// TIA Portal project "SemaforV1" (V15.1)

(* hardware
DEVICE "S71500/ET200MP station_1"  S7-1500 station
   slot 0: "Rail_0"  Rack  6ES7 590-1***0-0AA0
   slot 1: "PLC_1"  CPU 1513-1 PN  6ES7 513-1AL02-0AB0  V2.6
      slot 3: "CPU display_1"  6ES7591-1AA00-0AA0
DEVICE "HMI_1"  KTP900 Basic PN
   slot 0: "HMI_1"  KTP900 Basic PN  6AV2 123-2JB03-0AX0  15.1.0.0
   slot 1: "HMI_RT_1"  KTP900 Basic PN  6AV2 123-2JB03-0AX0  15.1.0.0
   slot 5: "HMI_1.IE_CP_1"  PROFINET Interface  15.0.1.0
      slot 1: "PROFINET Interface_1"  PROFINET Interface
         slot 1: "Port_1"  Port
*)

// ===== PLC "PLC_1"  CPU 1513-1 PN =====

VAR_GLOBAL   // PLC tag table "Default tag table"
   "Clock_Byte" AT %MB0 : Byte;
   "Clock_10Hz" AT %M0.0 : Bool;
   "Clock_5Hz" AT %M0.1 : Bool;
   "Clock_2.5Hz" AT %M0.2 : Bool;
   "Clock_2Hz" AT %M0.3 : Bool;
   "Clock_1.25Hz" AT %M0.4 : Bool;
   "Clock_1Hz" AT %M0.5 : Bool;
   "Clock_0.625Hz" AT %M0.6 : Bool;
   "Clock_0.5Hz" AT %M0.7 : Bool;
END_VAR

DATA_BLOCK "Semafor_Lumini"   // DB1
{ S7_Optimized_Access := 'TRUE' }
VERSION : 0.1
   VAR
      rosu_on : Bool;
      galben_on : Bool;
      verde_on : Bool;
      culoare_semafor : UInt;
      galben_intermitent_on : Bool;
   END_VAR
BEGIN
END_DATA_BLOCK

DATA_BLOCK "Semafor_Moduri"   // DB2
{ S7_Optimized_Access := 'TRUE' }
VERSION : 0.1
   VAR
      "mod_de functionare" : UInt;
      pornire_mod_normal : Bool;
      reseteaza_bucla : Bool;
      porneste_verde : Bool;
      porneste_galben : Bool;
      porneste_rosu : Bool;
      buton_pieton : Bool;
      timp_rosu : Time;
      Timp_galben : Time;
      timp_verde : Time;
      et_rosu : Time;
      et_galben : Time;
      et_verde : Time;
      timer_galben_hmi : Bool;
   END_VAR
BEGIN
END_DATA_BLOCK

DATA_BLOCK "Rising Edges"   // DB3
{ S7_Optimized_Access := 'TRUE' }
VERSION : 0.1
   VAR
      re1 : Bool;
      testing : Bool;
      "test count" : UInt;
   END_VAR
BEGIN
END_DATA_BLOCK

// folder: System blocks/Program resources

DATA_BLOCK "timer_verde"   // DB4
{ S7_Optimized_Access := 'TRUE' }
AUTHOR : Simatic
FAMILY : IEC
NAME : IEC_TMR
VERSION : 1.0
// stored: InstanceOfName IEC_TIMER
"IEC_TIMER"
BEGIN
END_DATA_BLOCK

DATA_BLOCK "timergalben"   // DB5
{ S7_Optimized_Access := 'TRUE' }
AUTHOR : Simatic
FAMILY : IEC
NAME : IEC_TMR
VERSION : 1.0
// stored: InstanceOfName IEC_TIMER
"IEC_TIMER"
BEGIN
END_DATA_BLOCK

DATA_BLOCK "timer rosu"   // DB6
{ S7_Optimized_Access := 'TRUE' }
AUTHOR : Simatic
FAMILY : IEC
NAME : IEC_TMR
VERSION : 1.0
// stored: InstanceOfName IEC_TIMER
"IEC_TIMER"
BEGIN
END_DATA_BLOCK

// folder: (top level)

ORGANIZATION_BLOCK "Main"   // OB1, LAD, ProgramCycle
TITLE = "Main Program Sweep (Cycle)"
{ S7_Optimized_Access := 'TRUE' }
VERSION : 0.1
   VAR_INPUT
      Initial_Call : Bool;   // Initial call of this OB
      Remanence : Bool;   // =True, if remanent data are available
   END_VAR
   VAR_TEMP   // added for the SCL form of the ladder/FBD networks
      _w1 : Bool;
   END_VAR
BEGIN

REGION Network 1: semafor modul normal
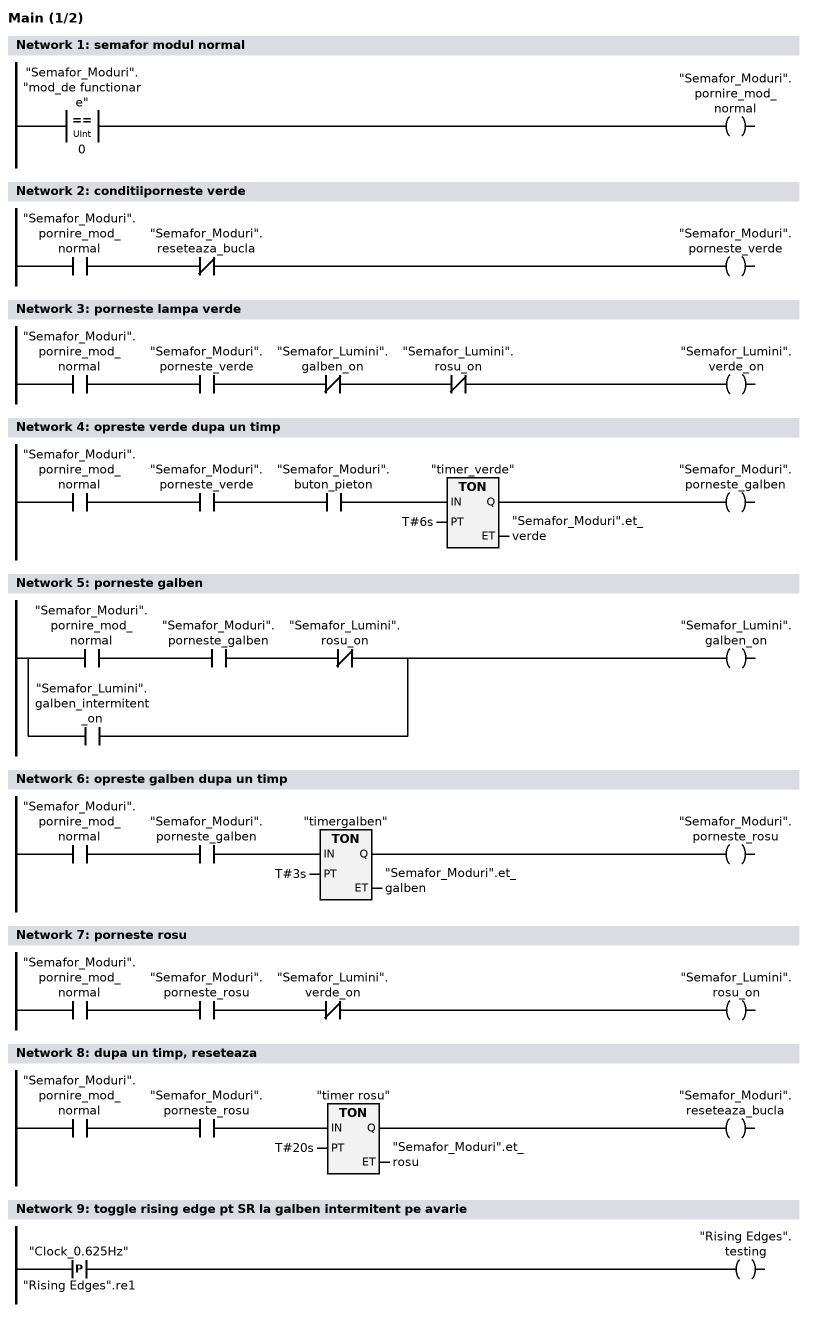
   RUNG wire#powerrail
      { S7_Templates := "SrcType := UInt" } EQ_Contact(in1 := "Semafor_Moduri"."mod_de functionare", in2 := 0)
      Coil( "Semafor_Moduri".pornire_mod_normal )
   END_RUNG
   // the same network as SCL:
   "Semafor_Moduri".pornire_mod_normal := "Semafor_Moduri"."mod_de functionare" = 0;
END_REGION

REGION Network 2: conditiiporneste verde
   RUNG wire#powerrail
      Contact( "Semafor_Moduri".pornire_mod_normal )
      I_Contact( "Semafor_Moduri".reseteaza_bucla )
      Coil( "Semafor_Moduri".porneste_verde )
   END_RUNG
   // the same network as SCL:
   "Semafor_Moduri".porneste_verde := "Semafor_Moduri".pornire_mod_normal AND NOT "Semafor_Moduri".reseteaza_bucla;
END_REGION

REGION Network 3: porneste lampa verde
   RUNG wire#powerrail
      Contact( "Semafor_Moduri".pornire_mod_normal )
      Contact( "Semafor_Moduri".porneste_verde )
      I_Contact( "Semafor_Lumini".galben_on )
      I_Contact( "Semafor_Lumini".rosu_on )
      Coil( "Semafor_Lumini".verde_on )
   END_RUNG
   // the same network as SCL:
   "Semafor_Lumini".verde_on := "Semafor_Moduri".pornire_mod_normal AND "Semafor_Moduri".porneste_verde AND NOT "Semafor_Lumini".galben_on AND NOT "Semafor_Lumini".rosu_on;
END_REGION

REGION Network 4: opreste verde dupa un timp
   "timer_verde".TON(IN := "Semafor_Moduri".pornire_mod_normal AND "Semafor_Moduri".porneste_verde AND "Semafor_Moduri".buton_pieton,
                     PT := T#6s,
                     ET => "Semafor_Moduri".et_verde);
   "Semafor_Moduri".porneste_galben := "timer_verde".Q;
END_REGION

REGION Network 5: porneste galben
   RUNG wire#powerrail
      Contact( "Semafor_Moduri".pornire_mod_normal )
      Contact( "Semafor_Moduri".porneste_galben )
      I_Contact( "Semafor_Lumini".rosu_on )
      wire#w1
      Coil( "Semafor_Lumini".galben_on )
   END_RUNG
   RUNG wire#powerrail
      Contact( "Semafor_Lumini".galben_intermitent_on )
   END_RUNG wire#w1
   // the same network as SCL:
   "Semafor_Lumini".galben_on := ("Semafor_Moduri".pornire_mod_normal AND "Semafor_Moduri".porneste_galben AND NOT "Semafor_Lumini".rosu_on) OR "Semafor_Lumini".galben_intermitent_on;
END_REGION

REGION Network 6: opreste galben dupa un timp
   "timergalben".TON(IN := "Semafor_Moduri".pornire_mod_normal AND "Semafor_Moduri".porneste_galben,
                     PT := T#3s,
                     ET => "Semafor_Moduri".et_galben);
   "Semafor_Moduri".porneste_rosu := "timergalben".Q;
END_REGION

REGION Network 7: porneste rosu
   RUNG wire#powerrail
      Contact( "Semafor_Moduri".pornire_mod_normal )
      Contact( "Semafor_Moduri".porneste_rosu )
      I_Contact( "Semafor_Lumini".verde_on )
      Coil( "Semafor_Lumini".rosu_on )
   END_RUNG
   // the same network as SCL:
   "Semafor_Lumini".rosu_on := "Semafor_Moduri".pornire_mod_normal AND "Semafor_Moduri".porneste_rosu AND NOT "Semafor_Lumini".verde_on;
END_REGION

REGION Network 8: dupa un timp, reseteaza
   "timer rosu".TON(IN := "Semafor_Moduri".pornire_mod_normal AND "Semafor_Moduri".porneste_rosu,
                    PT := T#20s,
                    ET => "Semafor_Moduri".et_rosu);
   "Semafor_Moduri".reseteaza_bucla := "timer rosu".Q;
END_REGION

REGION Network 9: toggle rising edge pt SR la galben intermitent pe avarie
   RUNG wire#powerrail
      P_Contact(operand := "Clock_0.625Hz", bit := "Rising Edges".re1)
      Coil( "Rising Edges".testing )
   END_RUNG
   // the same network as SCL:
   #_w1 := "Clock_0.625Hz" AND NOT "Rising Edges".re1;   // rising edge of "Clock_0.625Hz"
   "Rising Edges".re1 := "Clock_0.625Hz";
   "Rising Edges".testing := #_w1;
END_REGION

REGION Network 10: toggle test 2
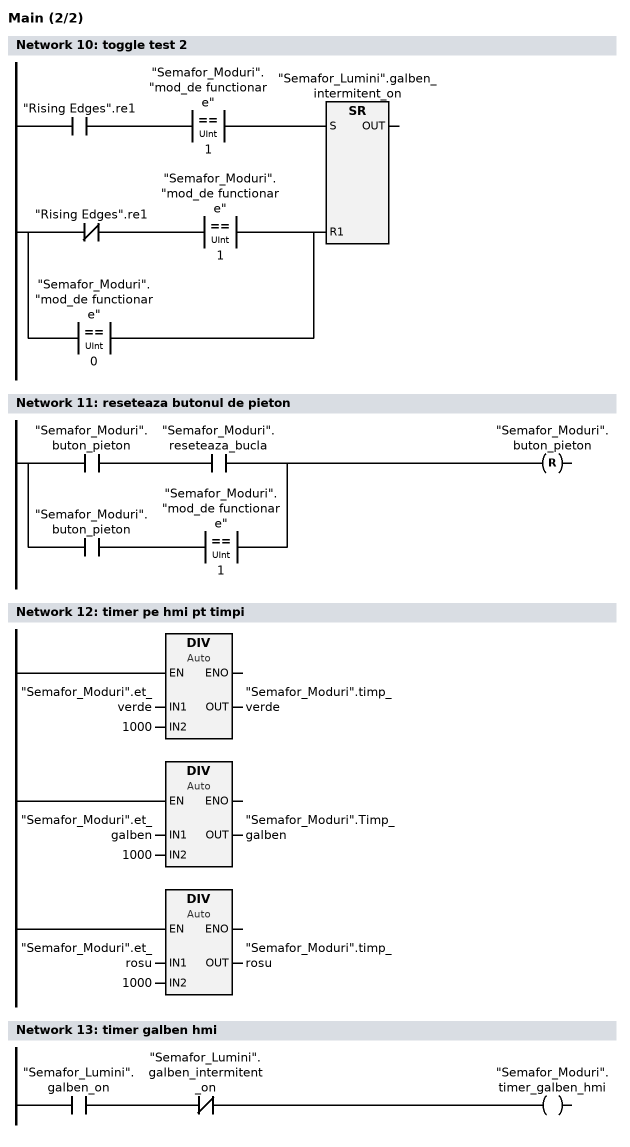
   RUNG wire#powerrail
      Contact( "Rising Edges".re1 )
      { S7_Templates := "SrcType := UInt" } EQ_Contact(in1 := "Semafor_Moduri"."mod_de functionare", in2 := 1)
      S_SR(operand := "Semafor_Lumini".galben_intermitent_on, r1 := wire#w1)
   END_RUNG
   RUNG wire#powerrail
      I_Contact( "Rising Edges".re1 )
      { S7_Templates := "SrcType := UInt" } EQ_Contact(in1 := "Semafor_Moduri"."mod_de functionare", in2 := 1)
   END_RUNG wire#w1
   RUNG wire#powerrail
      { S7_Templates := "SrcType := UInt" } EQ_Contact(in1 := "Semafor_Moduri"."mod_de functionare", in2 := 0)
   END_RUNG wire#w1
   // the same network as SCL:
   IF "Rising Edges".re1 AND ("Semafor_Moduri"."mod_de functionare" = 1) THEN
       "Semafor_Lumini".galben_intermitent_on := TRUE;   // SR flip-flop
   END_IF;
   IF (NOT "Rising Edges".re1 AND ("Semafor_Moduri"."mod_de functionare" = 1)) OR ("Semafor_Moduri"."mod_de functionare" = 0) THEN
       "Semafor_Lumini".galben_intermitent_on := FALSE;
   END_IF;
END_REGION

REGION Network 11: reseteaza butonul de pieton
   RUNG wire#powerrail
      Contact( "Semafor_Moduri".buton_pieton )
      Contact( "Semafor_Moduri".reseteaza_bucla )
      wire#w1
      R_Coil( "Semafor_Moduri".buton_pieton )
   END_RUNG
   RUNG wire#powerrail
      Contact( "Semafor_Moduri".buton_pieton )
      { S7_Templates := "SrcType := UInt" } EQ_Contact(in1 := "Semafor_Moduri"."mod_de functionare", in2 := 1)
   END_RUNG wire#w1
   // the same network as SCL:
   IF ("Semafor_Moduri".buton_pieton AND "Semafor_Moduri".reseteaza_bucla) OR ("Semafor_Moduri".buton_pieton AND ("Semafor_Moduri"."mod_de functionare" = 1)) THEN
       "Semafor_Moduri".buton_pieton := FALSE;
   END_IF;
END_REGION

REGION Network 12: timer pe hmi pt timpi
   RUNG wire#powerrail
      Div(in1 := "Semafor_Moduri".et_verde, in2 := 1000, out => "Semafor_Moduri".timp_verde)
   END_RUNG
   RUNG wire#powerrail
      Div(in1 := "Semafor_Moduri".et_galben, in2 := 1000, out => "Semafor_Moduri".Timp_galben)
   END_RUNG
   RUNG wire#powerrail
      Div(in1 := "Semafor_Moduri".et_rosu, in2 := 1000, out => "Semafor_Moduri".timp_rosu)
   END_RUNG
   // the same network as SCL:
   "Semafor_Moduri".timp_verde := "Semafor_Moduri".et_verde / 1000;
   "Semafor_Moduri".Timp_galben := "Semafor_Moduri".et_galben / 1000;
   "Semafor_Moduri".timp_rosu := "Semafor_Moduri".et_rosu / 1000;
END_REGION

REGION Network 13: timer galben hmi
   RUNG wire#powerrail
      Contact( "Semafor_Lumini".galben_on )
      I_Contact( "Semafor_Lumini".galben_intermitent_on )
      Coil( "Semafor_Moduri".timer_galben_hmi )
   END_RUNG
   // the same network as SCL:
   "Semafor_Moduri".timer_galben_hmi := "Semafor_Lumini".galben_on AND NOT "Semafor_Lumini".galben_intermitent_on;
END_REGION
END_ORGANIZATION_BLOCK

(* ===== HMI "HMI_RT_1" =====
system functions are stored by id; their names below are inferred from use
connection "HMI_Connection_1": ETHERNET, SMART_S7_1500_OMS

HMI tags "Default tag table"
   "Tag_ScreenNumber" : UInt, internal
   "Semafor_Moduri_mod_de functionare" : UInt = PLC Semafor_Moduri."mod_de functionare", 1 s
   "Semafor_Lumini_verde_on" : Bool = PLC Semafor_Lumini.verde_on, 1 s
   "Semafor_Lumini_galben_on" : Bool = PLC Semafor_Lumini.galben_on, 1 s
   "Semafor_Lumini_rosu_on" : Bool = PLC Semafor_Lumini.rosu_on, 1 s
   "Semafor_Moduri_buton_pieton" : Bool = PLC Semafor_Moduri.buton_pieton, 1 s
   "Semafor_Moduri_et_verde" : Time = PLC Semafor_Moduri.et_verde, 1 s
   "Semafor_Moduri_timp_verde" : Time = PLC Semafor_Moduri.timp_verde, 1 s
   "Semafor_Moduri_Timp_galben" : Time = PLC Semafor_Moduri.Timp_galben, 1 s
   "Semafor_Moduri_timp_rosu" : Time = PLC Semafor_Moduri.timp_rosu, 1 s
   "Semafor_Moduri_timer_galben_hmi" : Bool = PLC Semafor_Moduri.timer_galben_hmi, 1 s
   "Semafor_Lumini_galben_intermitent_on" : Bool = PLC Semafor_Lumini.galben_intermitent_on, 1 s

Template "Template_1" 800x480
   Button "Exit" at 722,440 size 55x39; TextOff 'Exit'; PictureOff "ExitRuntime_KTP900_Basic_PN_TR"; PictureOn "ExitRuntime_KTP900_Basic_PN_TR"
      on Release: StopRuntime(0)
   Button "Template_Button" at 622,440 size 55x39; TextOff 'Text'
   Button "Template_Button_1" at 522,440 size 55x39; TextOff 'Text'
   Button "Template_Button_2" at 422,440 size 55x39; TextOff 'Text'
   Button "Template_Button_3" at 322,440 size 55x39; TextOff 'Text'
   Button "Template_Button_4" at 222,440 size 55x39; TextOff 'Text'
   Button "Alarms" at 122,440 size 55x39; TextOff 'Alarms'; PictureOff "AlarmDisplay_KTP900_Basic_PN_TR"; PictureOn "AlarmDisplay_KTP900_Basic_PN_TR"
   Button "Start screen" at 22,440 size 55x39; TextOff 'Start screen'; PictureOff "NavigateHome_KTP900_Basic_PN_TR"; PictureOn "NavigateHome_KTP900_Basic_PN_TR"
      on Release: ActivateScreen("Root screen", 0)
   SymbolicIOField "Symbolic_IO_Field_Screen" at 73,7 size 620x26; TextOff '0'; TextOn '1'; TextList "TextList_ScreenNames"
      ProcessValue <- "Tag_ScreenNumber"
      on Change: ActivateScreenByNumber("Tag_ScreenNumber", 0)
   DateTimeField "HmiScreenItemData" at 695,20 size 105x20
   DateTimeField "HmiScreenItemData_1" at 695,0 size 105x20
   GraphicView "Logo" at 0,0 size 71x40; Picture "Logo of HMI_1"

screen "Root screen" 800x480, template "Template_1"
   on GenerateScreen: SetTag("Tag_ScreenNumber", 1)
   Circle "Circle_1" at 377,104 size 35x35
      Appearance <- "Semafor_Lumini_rosu_on"
   Circle "Circle_2" at 377,149 size 35x35
      Appearance <- "Semafor_Lumini_galben_on"
   Circle "Circle_3" at 377,194 size 35x35
      Appearance <- "Semafor_Lumini_verde_on"
   Button "Button_1" at 43,120 size 96x32; TextOff 'Pieton'
      on Click: SetTag("Semafor_Moduri_mod_de functionare", 0)
   Button "Button_2" at 43,172 size 96x32; TextOff 'Mod Avarie'
      on Click: SetTag("Semafor_Moduri_mod_de functionare", 1)
   Button "Button_3" at 43,224 size 96x32; TextOff 'Buton Pieton'
      on Click: SetBit("Semafor_Moduri_buton_pieton")
   IOField "I/O field_1" at 575,72 size 96x32; FormatPattern 9999; Unit s
      Visibility <- "Semafor_Lumini_verde_on"
      ProcessValue <- "Semafor_Moduri_timp_verde"
   IOField "I/O field_2" at 575,72 size 96x32; FormatPattern 9999; Unit s
      ProcessValue <- "Semafor_Moduri_Timp_galben"
      Visibility <- "Semafor_Moduri_timer_galben_hmi"
   IOField "I/O field_3" at 575,72 size 96x32; FormatPattern 9999; Unit s
      ProcessValue <- "Semafor_Moduri_timp_rosu"
      Visibility <- "Semafor_Lumini_rosu_on"
   TextField "Text field_1" at 30,39 size 331x25; Text 'Semafor intermitent, circulati cu grija!'
      Visibility <- "Semafor_Moduri_mod_de functionare"
*)